// SIMATIC S7-200 project (STEP 7-Micro/WIN), CPU 224XP REL 02.01

SYMBOL_TABLE USUARIO1
MARCHA           I0.0
PARO             I0.1
LAMPARA1         Q0.0
LAMPARA2         Q0.1
END_SYMBOL_TABLE

ORGANIZATION_BLOCK PRINCIPAL:OB1
TITLE=COMENTARIOS DEL PROGRAMA
BEGIN
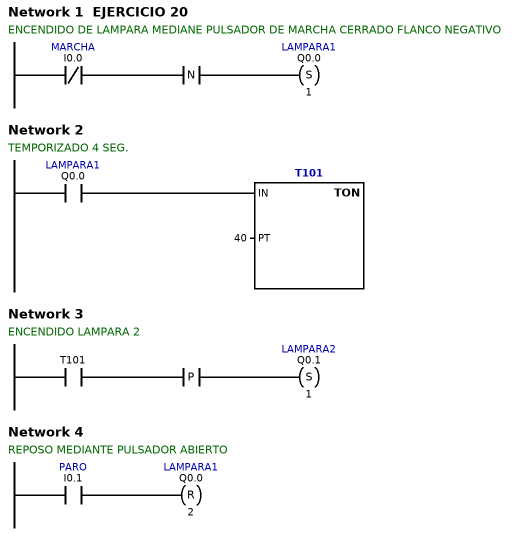
Network 1 // EJERCICIO 20
// ENCENDIDO DE LAMPARA MEDIANE PULSADOR DE MARCHA CERRADO FLANCO NEGATIVO 
// (network saved uncompiled; LAD cells follow)
// row 0: c0 -|/|- MARCHA:I0.0  c1 -|N|-  c2 -(S) LAMPARA1:Q0.0, 1
Network 2
// TEMPORIZADO 4 SEG. 
LD     LAMPARA1:Q0.0
TON    T101, 40
Network 3
// ENCENDIDO LAMPARA 2 
// (network saved uncompiled; LAD cells follow)
// row 0: c0 -| |- T101  c1 -|P|-  c2 -(S) LAMPARA2:Q0.1, 1
Network 4
// REPOSO MEDIANTE PULSADOR ABIERTO 
LD     PARO:I0.1
R      LAMPARA1:Q0.0, 2
END_ORGANIZATION_BLOCK
